FUNCTION_BLOCK TcoRemoteTaskTestContext EXTENDS TcoCore._internals_TcoContext
VAR
	_sut : TcoRemoteTaskTest(THIS^, NO.Structure);
    _invokeInitializedCSharpMethodDone : BOOL;
    _invokeNotInitializedCSharpMethodDone : BOOL;
    _exceptionInMethodWillResultInExceptionDone : BOOL;
	_sharedVariable : INT;
	
END_VAR

METHOD PROTECTED Main

CASE _testId OF
    0:
        _invokeInitializedCSharpMethodDone := FALSE;
        _invokeNotInitializedCSharpMethodDone := FALSE;
        _exceptionInMethodWillResultInExceptionDone := FALSE;
    eTcoRemoteTaskTests.RestoreTasks:
        _sut._invokeInitializedCSharpMethod.Restore();
        _sut._invokeNotInitializedCSharpMethod.Restore();
        _sut._exceptionInMethodWillResultInException.Restore();
    eTcoRemoteTaskTests.InvokeInitializedCSharpMethod:
        _invokeInitializedCSharpMethodDone := _sut._invokeInitializedCSharpMethod.Invoke().Done;
    eTcoRemoteTaskTests.InvokeNotInitializedCSharpMethod:
        _invokeNotInitializedCSharpMethodDone := _sut._invokeNotInitializedCSharpMethod.Invoke().Error;
    eTcoRemoteTaskTests.ExceptionInMethodWillResultInException:
        _exceptionInMethodWillResultInExceptionDone := _sut._exceptionInMethodWillResultInException.Invoke().Error;
END_CASE

_sut();
END_METHOD

END_FUNCTION_BLOCK

(* stored: Version 1.1.0.1
   POU TcoRemoteTaskTestContext: Id {e0205570-0107-044a-09e9-3ba686b39cfb}, SpecialFunc None
   Method Main: Id {726bdbc0-118a-02d2-27eb-5048fd798ca9} *)
